TYPE CmpConvBreakStopGroup :
STRUCT
	Framework: Framework;
	ConvRunning: ARRAY[1..cBreakStopGroupMaxInstance] OF BOOL;
	LowerStopReq: ARRAY[1..cBreakStopGroupMaxInstance] OF BOOL;
	Config: CmpConvBreakStopGroupConfig;
END_STRUCT
END_TYPE

(* stored: Version 1.1.0.1, ProductVersion 3.1.4024.6
   DUT CmpConvBreakStopGroup: Id {5416f3ac-39b5-4b49-a4b8-bc9c02a83f24} *)
